{region '#Template'}
	{attribute 'Version' := '5.0.0.0'}
	{attribute 'Tags' := '"LCID": "1031", "Text": "Universal, Control, Event class, Notification"'}
	{attribute 'Tags' := '"LCID": "1033", "Text": "Universal, Control, Event class, Notification"'}
	{attribute 'Using' := '"Type": "Template", "URI": "EC_ID"'}
	{attribute 'Description' := '"LCID": "1031", "Text": "Ereignisklasse"'}
	{attribute 'Description' := '"LCID": "1033", "Text": "Event class"'}
{endregion}
FUNCTION_BLOCK FB_BA_EvtCategory EXTENDS FB_BA_View
VAR_INPUT CONSTANT
		EC				: FB_BA_EC;  
END_VAR

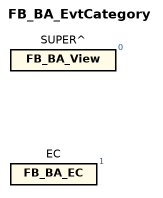
SUPER^(); // FB_BA_View
EC(); // FB_BA_EC

METHOD FB_init : BOOL
VAR_INPUT
	bInitRetains : BOOL; // if TRUE, the retain variables are initialized (warm start / cold start)
	bInCopyCode : BOOL;  // if TRUE, the instance afterwards gets moved into the copy code (online change)
END_VAR
EC.iParent					:= THIS^;
EC.iLabel					:= LblCtl_EvtClass;   
EC.nInstanceID				:= EC_ID.NC10;
EC.eEventType				:= E_BA_EventType.eAlarm;
EC.aPriority[1]				:= 16;
EC.aPriority[2]				:= 17;
EC.aPriority[3]				:= 18;
END_METHOD

END_FUNCTION_BLOCK

(* stored: Version 1.1.0.1, ProductVersion 3.1.4024.12
   POU FB_BA_EvtCategory: Id {72befd9f-8de7-4529-bbe8-4fb44b0c594d}, SpecialFunc None
   Method FB_init: Id {6c3def9f-31e6-4b16-b806-67db1f99dcb0} *)
